// TwinCAT 3 PLC project PRG_B_Actuator
// Title: B_Actuator
// Company: RafalOS
// Author: Rafał Osajda
// ProjectVersion: 0.0.0.4
// ProgramVersion: 3.1.4024.0
// libraries:
//   B_Base, * (RafalOS)
//   B_IO, * (RafalOS)
//   Tc2_Standard, * (Beckhoff Automation GmbH)
//   Tc2_System, * (Beckhoff Automation GmbH)
//   Tc3_Module, * (Beckhoff Automation GmbH)
// project tree:
//   / PlcTask.TcTTO (not stored)
//   POUs Compilation/ PRG_Compilation.TcPOU (not stored)
//   POUs/ FB_Actuator.TcPOU (not stored), ITF_Actuator.TcIO, ITF_Actuator_HMI_Command.TcIO, ITF_Actuator_HMI_Init.TcIO, ITF_Actuator_HMI_Connector.TcIO

// ---- POUs/ITF_Actuator.TcIO
INTERFACE ITF_Actuator EXTENDS ITF_BaseControlElement

METHOD IsEnd : BOOL
VAR_INPUT
END_VAR
END_METHOD

METHOD PUBLIC IsStart : BOOL
VAR_INPUT
END_VAR
END_METHOD

(*			
	EVERDE sp. z o.o.
	Rafał Osajda		31.03.2025		TC 4024.66
	Uruchomienie cyklu przesuwania do początku
*)
METHOD PUBLIC MoveToEnd
VAR_INPUT
END_VAR
END_METHOD

(*			
	EVERDE sp. z o.o.
	Rafał Osajda		31.03.2025		TC 4024.66
	Uruchomienie cyklu przesuwania do początku
*)
METHOD PUBLIC MoveToStart
VAR_INPUT
END_VAR
END_METHOD

METHOD PUBLIC MovingToEndBusy : BOOL
VAR_INPUT
END_VAR
END_METHOD

METHOD PUBLIC MovingToEndFirstCycyle : BOOL
VAR_INPUT
END_VAR
END_METHOD

METHOD PUBLIC MovingToEndStatus : BOOL
VAR_INPUT
END_VAR
END_METHOD

METHOD PUBLIC MovingToStartBusy : BOOL
VAR_INPUT
END_VAR
END_METHOD

METHOD PUBLIC MovingToStartFirstCycle : BOOL
VAR_INPUT
END_VAR
END_METHOD

METHOD PUBLIC MovingToStartStatus : BOOL
VAR_INPUT
END_VAR
END_METHOD

END_INTERFACE

// ---- POUs/ITF_Actuator_HMI_Command.TcIO
INTERFACE ITF_Actuator_HMI_Command

(*			
	EVERDE sp. z o.o.
	Rafał Osajda		31.03.2025		TC 4024.66
	Uruchomienie cyklu przesuwania do początku
*)
METHOD PUBLIC MoveToEnd
VAR_INPUT
END_VAR
END_METHOD

(*			
	EVERDE sp. z o.o.
	Rafał Osajda		31.03.2025		TC 4024.66
	Uruchomienie cyklu przesuwania do początku
*)
METHOD PUBLIC MoveToStart
VAR_INPUT
END_VAR
END_METHOD

END_INTERFACE

// ---- POUs/ITF_Actuator_HMI_Init.TcIO
INTERFACE ITF_Actuator_HMI_Init EXTENDS ITF_BaseControlElement, ITF_Actuator_HMI_Connector, ITF_Actuator_HMI_Command

END_INTERFACE

// ---- POUs/ITF_Actuator_HMI_Connector.TcIO
INTERFACE ITF_Actuator_HMI_Connector EXTENDS ITF_BaseControlElement_HMI_Connector

METHOD GetTimeLastMove : TIME
VAR_INPUT
END_VAR
END_METHOD

METHOD IsEnd : BOOL
VAR_INPUT
END_VAR
END_METHOD

METHOD PUBLIC IsStart : BOOL
VAR_INPUT
END_VAR
END_METHOD

METHOD PUBLIC MovingToEndBusy : BOOL
VAR_INPUT
END_VAR
END_METHOD

METHOD PUBLIC MovingToEndStatus : BOOL
VAR_INPUT
END_VAR
END_METHOD

METHOD PUBLIC MovingToStartBusy : BOOL
VAR_INPUT
END_VAR
END_METHOD

METHOD PUBLIC MovingToStartStatus : BOOL
VAR_INPUT
END_VAR
END_METHOD

END_INTERFACE
